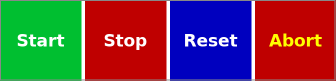
VISUALIZATION VFM_MachineControl  // 336x81
VAR_IN_OUT
	HMI: ST_HMI_Machine;
END_VAR
    Rectangle (0,0 81x81), "Start"
        tap HMI.Command.Start
    Rectangle (85,0 81x81), "Stop"
        tap HMI.Command.Stop
    Rectangle (170,0 81x81), "Reset"
        tap HMI.Command.Reset
    Rectangle (255,0 81x81), "Abort"
        toggle HMI.Command.Abort
END_VISUALIZATION

(* stored: Version 1.1.0.1, ProductVersion 3.1.4024.12
   Visu VFM_MachineControl: Id {77d0dbab-0ecf-4bad-af16-66583414dfce} *)
